FUNCTION_BLOCK FB_AUT_145 EXTENDS FB_AUT_ABSTRACT
(****************************************************************************)
(*	POU_AUT_zxx			Bausteinaufrufe Station	zxx							*)
(*	Status				ungetestet											*)
(*  Version:			1.0													*)
(*	Beschrieb:																*)
(*																			*)
(*	Abläufe:			FB_ABLzxxA		Hauptablauf							*)
(*																			*)
(*																			*)
(* 	25.09.2019/Dj															*)
(****************************************************************************)
(*	dd.mm.yyyy   KZ    x.y			Beschrieb								*)
(****************************************************************************)
VAR_INPUT
    (* spezifische Eingänge *)

END_VAR
VAR_OUTPUT
    (* spezifische Ausgänge *)

END_VAR
VAR
    (* Bausteine *)
    fb_Pnp    : FB_ABL_145_Pnp;
    fb_Feeder : FB_ABL_145_Feeder;

    fb_stat_pnp    : FB_AUT_Statistics;
    fb_stat_Feeder : FB_AUT_Statistics;

END_VAR

VAR CONSTANT
    ROT_TABLE_FREE_MAX_Y : REAL := 100.0; // If Y and Z axis is more than this value, the feeder cannot move
    ROT_TABLE_FREE_MAX_Z : REAL := 50.0; // If Z and Y axis is more than this value, the feeder cannot move

    PNP_VERTICAL_MAX_Z : REAL := 50.0; // If Z axis is more than this value, the horizontal axis of the pnp cannot move
END_VAR

(*******************************************************************)
(* Timer *)
(*******************************************************************)

(*******************************************************************)
(* Flanken / Merker *)
(*******************************************************************)
//MANU CYCLE
IF (enIN_State = StateMANU) AND xIN_ManuCycle THEN
    xManuCycle := TRUE;
END_IF;

IF (enIN_State <> StateMANU) OR xOUT_Done THEN
    xManuCycle := FALSE;
END_IF

//NEXT STEP
xNextStep := (enIN_State > StateSTEP) OR
             ((enIN_State = StateSTEP) AND xIN_Step) OR
             ((enIN_State = StateMANU) AND xManuCycle);

//RESET
xReset := (enIN_State < StateREADY) AND (enIN_State <> StateINIT) AND NOT xManuCycle;

(*******************************************************************)
(* Bausteinaufrufe Abläufe *)
(*******************************************************************)

xRelease := MAIN.MoverMan.IsProcessUsed(THIS^);

fb_Pnp(xIN_Reset          := xReset,
       xIN_Init           := xIN_Init,
       xIN_Quit           := xIN_Quit,
       xIN_Start          := enIN_State >= enState.StateLEER AND xRelease,
       xIN_Sperre         := NOT xIN_On,
       xIN_NextStep       := xNextStep,
       xIN_AlarmAktiv     := xIN_AlarmAktiv,
       xIN_DryCycle       := xIN_DryCycle,
       xIN_RestartCYCL    := enIN_State >= enState.StateLEER,
       enIN_State         := enIN_State,
       tIN_Timeout        := tIN_Timeout,
       pxFG_Freigabe      := ADR(xRelease),
       Mover              := THIS^.Mover,
       xIN_PceReadyToPick := fb_Feeder.xOUT_Done,
       xIN_HorAxisFree    := ST145_Axis.axis145_02Z.rActPos < ROT_TABLE_FREE_MAX_Y);

fb_Feeder(xIN_Reset       := xReset,
          xIN_Init        := xIN_Init,
          xIN_Quit        := xIN_Quit,
          xIN_Start       := enIN_State >= enState.StateLEER AND xRelease,
          xIN_Sperre      := NOT xIN_On,
          xIN_NextStep    := xNextStep,
          xIN_AlarmAktiv  := xIN_AlarmAktiv,
          xIN_DryCycle    := xIN_DryCycle,
          xIN_RestartCYCL := enIN_State >= enState.StateLEER,
          enIN_State      := enIN_State,
          tIN_Timeout     := tIN_Timeout,
          pxFG_Freigabe   := ADR(xRelease),
          // special
          xIN_PickPiece            := fb_Pnp.xOUT_PickPiece,
          xIN_RotTableBlockedByPnp := (ST145_Axis.axis145_01Y.rActPos > ROT_TABLE_FREE_MAX_Y) AND
                                      (ST145_Axis.axis145_02Z.rActPos > ROT_TABLE_FREE_MAX_Z));

fb_stat_pnp(xIN_Enable  := enState.StateAUTO = enIN_State,
            xIN_Waiting := fb_Pnp.xOUT_Wait,
            xIN_Running := (fb_Pnp.iOUT_Step >= ST145_Pnp_e.START) AND
                           (fb_Pnp.iOUT_Step <= ST145_Pnp_e.DONE),
            // Since we use a mover system, a cycle is done when we are waiting on a mover
            xIN_Done := fb_Pnp.iOUT_Step = ST145_Pnp_e.waitOnMover);

fb_stat_Feeder(xIN_Enable  := enState.StateAUTO = enIN_State,
               xIN_Waiting := fb_feeder.xOUT_Wait,
               xIN_Running := (fb_feeder.iOUT_Step >= ST145_Feeder_e.START) AND
                              (fb_feeder.iOUT_Step <= ST145_Feeder_e.DONE),
               xIN_Done := fb_feeder.iOUT_Step = ST145_Feeder_e.DONE);

(*******************************************************************)
(* Mover reset flags *)
(*******************************************************************)

(*******************************************************************)
(* OUTPUT *)
(*******************************************************************)
xOUT_InitDone := fb_Pnp.xOUT_InitDone AND fb_Feeder.xOUT_InitDone;
xOUT_Ready    := fb_Pnp.xOUT_Ready AND fb_Feeder.xOUT_Ready;
xOUT_Done     := fb_Pnp.xOUT_Done; // we ignore feeder
xOUT_ErrFlag  := fb_Pnp.xOUT_ErrFlag OR fb_Feeder.xOUT_ErrFlag;
xOUT_Wait     := fb_Pnp.xOUT_Wait AND fb_Feeder.xOUT_Wait;
xOUT_AlarmST  := xOUT_ErrFlag;

(*******************************************************************)
(* Bausteinaufruf Error Station *)
(*******************************************************************)
// POU_ERR_VORLAGE(xIN_QUIT:=xIN_Quit , pstrArIN_ALARM:=ADR(HMI.strArALARM[1]));

(* % of completion of the process *)
PROPERTY iCompletionPC : INT
GET
iCompletionPC := THIS^.fb_Pnp.iOUT_ProcessCompletion;
END_GET
END_PROPERTY

PROPERTY ProcessExecution : ProcessExecution_e
GET
ProcessExecution := THIS^._ProcessExecution;
END_GET
SET
THIS^._ProcessExecution := ProcessExecution;
END_SET
END_PROPERTY

PROPERTY xBusy : BOOL
GET
xBusy := THIS^.fb_Pnp.xOUT_Busy;
END_GET
SET
END_SET
END_PROPERTY

PROPERTY xDone : BOOL
GET
xDone := THIS^.fb_Pnp.xOUT_Ready OR THIS^.fb_Pnp.xOUT_Done;
END_GET
END_PROPERTY

PROPERTY xMoverPathFree : BOOL
GET
xMoverPathFree := THIS^.fb_Pnp.xOUT_MoverFree OR THIS^.fb_Pnp.xOUT_Ready OR THIS^.fb_Pnp.xOUT_Done;
END_GET
END_PROPERTY

PROPERTY xMoverShouldLeave : BOOL
GET
xMoverShouldLeave := THIS^.fb_Pnp.iOUT_Step = ST145_Pnp_e.SYNC_MOVER_LEAVE;
END_GET
END_PROPERTY

END_FUNCTION_BLOCK

(* stored: Version 1.1.0.1, ProductVersion 3.1.4024.6
   POU FB_AUT_145: Id {08112b02-0fc6-41b6-9857-0e54cdf1e202}, SpecialFunc None
   Property iCompletionPC: Id {2942a88c-0ac7-4907-9545-bc0952d0bbd4}
   Get Get: Id {f5810122-27f0-44a4-9ec6-52e1cce8a9c9}
   Property ProcessExecution: Id {261c9f48-b1f0-42c4-ac0f-b536dde8972d}
   Get Get: Id {868d144b-9382-4ae6-8c78-a569fa6ff24f}
   Set Set: Id {15cc1ab5-5aa8-4b19-b117-a9ddd2ec1c7f}
   Property xBusy: Id {730bba88-5429-4a81-a9c8-f30622e992d1}
   Get Get: Id {3a3e7614-8191-46d6-b8a4-9f7b51dacf61}
   Set Set: Id {d54be088-acdd-4f28-8320-c91983b74d4d}
   Property xDone: Id {c3d01f69-afbd-4593-9872-d9731c6a5021}
   Get Get: Id {ae7577b2-703d-412c-95bb-41f265fcd48b}
   Property xMoverPathFree: Id {d0820e50-9284-4095-beba-0a0740a2906e}
   Get Get: Id {6e549b05-1759-4f68-b59b-e80a30e93eae}
   Property xMoverShouldLeave: Id {f177a4fc-7b15-41ec-94d1-7ea05a42e1da}
   Get Get: Id {1889b387-c08f-4995-9f37-6c15116b8121} *)
